PROGRAM MAIN_Receiver
VAR
	// SMPTE Receiver
	SMPTE_Receiver 	: FB_SMPTE_Receiver;
	ReceivingSignal	: BOOL;
	FrameRate		: REAL;
	TimeString		: STRING;
	TimeStruct		: ST_SMPTE_TimeStruct;
END_VAR

(************************)
(**** SMPTE Receiver ****)
(************************)

// Call the execute method once each cycle
SMPTE_Receiver.Cycle();
// Check if the cable is connected and receiving timecode analog signal
ReceivingSignal := SMPTE_Receiver.Receiving;
// Get the framerate
FrameRate := SMPTE_Receiver.FrameRate;
// Get the time as string output
TimeString := SMPTE_Receiver.TimeString;
// Get the time as time struct
TimeStruct := SMPTE_Receiver.TimeStruct;

END_PROGRAM

(* stored: Version 1.1.0.1, ProductVersion 3.1.4024.12
   POU MAIN_Receiver: Id {829cf880-89e0-4808-9386-f68ae7048a02}, SpecialFunc None *)
